Fanuc TP program (LS listing): COPYPR.LS

/PROG  COPYPR
/ATTR
OWNER		= MNEDITOR;
COMMENT		= "";
PROG_SIZE	= 195;
CREATE		= DATE 30-06-13  TIME 04:12:40;
MODIFIED	= DATE 31-08-01  TIME 05:38:36;
FILE_NAME	= ;
VERSION		= 0;
LINE_COUNT	= 2;
MEMORY_SIZE	= 559;
PROTECT		= READ_WRITE;
TCD:  STACK_SIZE	= 0,
      TASK_PRIORITY	= 50,
      TIME_SLICE	= 0,
      BUSY_LAMP_OFF	= 0,
      ABORT_REQUEST	= 0,
      PAUSE_REQUEST	= 0;
DEFAULT_GROUP	= 1,*,*,*,*;
CONTROL_CODE	= 00000000 00000000;
/APPL
/APPL

AUTO_SINGULARITY_HEADER;
  ENABLE_SINGULARITY_AVOIDANCE   : TRUE;
/MN
   1:  PR[211:Styl Load 15533]=PR[123:Styl Load 533]    ;
   2:  PR[151:Styl Unld 15533]=PR[133:Styl Unload 533]    ;
/POS
/END
